// TIA Portal V17 export
VAR_GLOBAL   // PLC tag table "Tags_Caldeira"
   Botao_liga AT %I0.0 : Bool;   // Botao de impulso para partida do sistema (NA)
   Botao_desliga AT %I0.1 : Bool;   // Botao de impulso para parada natural (NF)
   Botao_reset AT %I0.2 : Bool;   // Botao de impulso para reconhecimento de falha (NF)
   Botao_emergencia AT %I0.3 : Bool;   // Botao cogumelo de parada imediata (NF com retencao)
   AI_Nivel AT %IW64 : Int;   // Leitura analogica de nivel do reservatorio (4-20mA)
   AI_Pressao AT %IW66 : Int;   // Leitura analogica de pressao interna do cilindro (4-20mA)
   AI_Temperatura AT %IW68 : Int;   // Leitura analogica de temperatura interna do trocador (4-20mA)
   Valvula_Agua AT %Q0.0 : Bool;   // Valvula ON/OFF de abastecimento continuo de agua
   Valvula_Vapor AT %Q0.1 : Bool;   // Valvula principal de vapor para linha de producao
   Valvula_Alivio AT %Q0.2 : Bool;   // Valvula de alivio rapido de sobrepressao e emergencia
   Queimador_1 AT %Q0.3 : Bool;   // Acionamento do Queimador 1
   Queimador_2 AT %Q0.4 : Bool;   // Acionamento do Queimador 2
   Queimador_3 AT %Q0.5 : Bool;   // Acionamento do Queimador 3
   Queimador_4 AT %Q0.6 : Bool;   // Acionamento do Queimador 4
   Queimador_5 AT %Q0.7 : Bool;   // Acionamento do Queimador 5
   Queimador_6 AT %Q1.0 : Bool;   // Acionamento do Queimador 6
   Lamp_Sistema_Lig AT %Q1.1 : Bool;   // Sinalizacao luminosa: Sistema em operacao
   Lamp_Alarme_Emerg AT %Q1.2 : Bool;   // Sinalizacao luminosa: Alarme de Emergencia ativado
END_VAR
